TYPE EtcMasterBase_62654B43 :
STRUCT
END_STRUCT
END_TYPE

(* stored: Version 1.2.0.0, ProductVersion 3.1.4024.9
   DUT EtcMasterBase_62654B43: Id {c5342aa5-8fdf-4fcb-b45b-1a5283326192} *)
